FUNCTION_BLOCK EquipmentModule EXTENDS FB_PackML_BaseModule
VAR_INPUT
END_VAR
VAR_OUTPUT
END_VAR
VAR
END_VAR

END_FUNCTION_BLOCK

(* stored: Version 1.1.0.1, ProductVersion 3.1.4024.12
   POU EquipmentModule: Id {2e44d4e8-09ab-435d-a0e1-458f7bc1a6a4}, SpecialFunc None *)
